{attribute 'qualified_only'}
VAR_GLOBAL
	program_state : state_enum;
END_VAR

(* stored: Version 1.1.0.1, ProductVersion 3.1.4024.13
   GVL Global_Variables: Id {232f4ff8-114a-48eb-8680-bd949f3079f0} *)
